TYPE "bioSig.DT"
TITLE = Batch I/O Signal Data Type
// -- Woermann Automation --
AUTHOR : Woermann
VERSION : 0.1
	STRUCT
		Sig :  Bool;   // (O) Signal
		_Sig :  Bool;   // (O) Internal Signal
		Raw : Bool;   // (I) Raw Signal
		Res : Bool;   // (I) Reset Signal (Latched Type)
		Set { S7_SetPoint := 'True'} :  Bool;   // (I) Required Setting of Signal (Sig)

		Typ : Byte;   // (I) Type

		OnTSetP { S7_SetPoint := 'True'} : Real;   // (I) On Time Delay Setpoint
		OnTVal : Real := 0.0;   // (I/O) On Time Delay Value
		OffTSetP { S7_SetPoint := 'True'} : Real;   // (I) Off Time Delay Setpoint
		OffTVal : Real := 0.0;   // (I/O) Off Time Delay Value

		Off :  Bool;   // (O) Off / Closed (dark grey)
		On :  Bool;   // (O) On / Open (light green)
		MOff :  Bool;   // (O) Moving to Off / Closing (light grey)
		MOn :  Bool;   // (O) Moving to On / Opening (dark green)

		Alm :  Bool;   // (O) Alarm
		AlmS :  Bool;   // (O) Alarm Saved (Not Ackknowledged)
		EAlm { S7_SetPoint := 'True'} :  Bool;   // (I) Enable Alarm Evaluation
		AlmTSetP { S7_SetPoint := 'True'} : Real := 10.0;   // (I) Alarm Time Delay Setpoint
		AlmTVal : Real := 0.0;   // (I/O) Alarm Time Delay
		Wrn :  Bool;   // (O) Warning
		EWrn { S7_SetPoint := 'True'} :  Bool;   // (I) Enable Warning Evaluation
	END_STRUCT;

END_TYPE

